# EPICS substitutions: iocs/example/labApp/Db/lab_expanded.substitutions
# This file was automatically generated on Fri 25 May 2018 08:06:14 BST from
# source: /home/hgv27681/R3.14.12.3/support/pmac/etc/makeIocs/lab.xml
#
# *** Please do not edit this file: edit the source file instead. ***
#

# Macros:
#  PORT      The asyn port for the pmac controller
#  P         PV Prefix
#  NAXES     Number of axes
#  TIMEOUT   Timeout for controller communication
#  FEEDRATE  feedrate below which we go into error
#  CSG0      Name for Coordinate System Group 0
#  CSG1      Name for Coordinate System Group 1
#  CSG2      Name for Coordinate System Group 2
#  CSG3      Name for Coordinate System Group 3
#  CSG4      Name for Coordinate System Group 4
#  CSG5      Name for Coordinate System Group 5
#  CSG6      Name for Coordinate System Group 6
#  CSG7      Name for Coordinate System Group 7
file $(PMAC)/db/pmacController.template
{
pattern { PORT, P, NAXES, TIMEOUT, FEEDRATE, CSG0, CSG1, CSG2, CSG3, CSG4, CSG5, CSG6, CSG7 }
    { "Brick", "BRICK1", "8", "4", "100", "1,2->A,B", "3,4->I", "MIXED CS3", "MIXED CS2", "", "", "", "" }
}

# Macros:
#  PORT  The asyn port for the pmac controller
#  P     PV Prefix
# For Non-Power PMAC, use pmacStatus.template instead
file $(PMAC)/db/powerPmacStatus.template
{
pattern { PORT, P }
    { "Brick", "BRICK1" }
}

# Macros:
#  PMAC  Pmac/Geobrick name
#  AXIS  Axis number
#  PORT  Asyn port
file $(PMAC)/db/pmacStatusAxis.template
{
pattern { PMAC, AXIS, PORT }
    { "BRICK1", "1", "Brick" }
    { "BRICK1", "2", "Brick" }
    { "BRICK1", "3", "Brick" }
    { "BRICK1", "4", "Brick" }
    { "BRICK1", "5", "Brick" }
    { "BRICK1", "6", "Brick" }
    { "BRICK1", "7", "Brick" }
    { "BRICK1", "8", "Brick" }
}

# Macros:
#  P                Device Prefix
#  M                Device Suffix
#  PORT             Delta tau motor controller
#  ADDR             Address on controller
#  DESC             Description, displayed on EDM screen
#  MRES             Motor Step Size (EGU)
#  VELO             Velocity (EGU/s)
#  PREC             Display Precision
#  EGU              Engineering Units
#  TWV              Tweak Step Size (EGU)
#  DTYP             DTYP of record
#  DIR              User Direction
#  VBAS             Base Velocity (EGU/s)
#  VMAX             Max Velocity (EGU/s), defaults to VELO
#  ACCL             Seconds to Velocity
#  BDST             BL Distance (EGU)
#  BVEL             BL Velocity (EGU/s)
#  BACC             BL Seconds to Veloc.
#  DHLM             Dial High Limit
#  DLLM             Dial Low Limit
#  HLM              User High Limit
#  LLM              User Low Limit
#  HLSV             HW Lim. Violation Svr
#  INIT             Startup commands
#  SREV             Steps per Revolution
#  RRES             Readback Step Size (EGU)
#  ERES             Encoder Step Size (EGU)
#  JAR              Jog Acceleration (EGU/s^2)
#  UEIP             Use Encoder If Present
#  URIP             Use RDBL If Present
#  RDBL             Readback Location, set URIP = 1 if you specify this
#  RLNK             Readback output link
#  RTRY             Max retry count
#  DLY              Readback settle time (s)
#  OFF              User Offset (EGU)
#  RDBD             Retry Deadband (EGU)
#  FOFF             Freeze Offset, 0=variable, 1=frozen
#  ADEL             Alarm monitor deadband (EGU)
#  NTM              New Target Monitor, only set to 0 for soft motors
#  FEHIGH           HIGH limit for following error
#  FEHIHI           HIHI limit for following error
#  FEHHSV           HIHI alarm severity for following error
#  FEHSV            HIGH alarm severity for following error
#  SCALE            Scale factor, if pmacSetAxisScale is used this should be set
#  HOMEVIS          If 1 then home is visible on the gui
#  HOMEVISSTR       If HOMEVIS=0, then display this text on the gui instead
#  name             Object name and gui association name
#  alh              Set this to alh to add the motor to the alarm handler and send emails,
#  gda_name         Name to export this as to GDA
#  gda_desc         Description to export this as to GDA
#  SPORT            Delta tau motor controller comms port
#  HOME             Prefix for autohome instance. Defaults to $(P). If unspecified,
#  ALLOW_HOMED_SET  Set to a blank to allow this axis to have its homed
file $(PMAC)/db/dls_pmac_asyn_motor.template
{
pattern { P, M, PORT, ADDR, DESC, MRES, VELO, PREC, EGU, TWV, DTYP, DIR, VBAS, VMAX, ACCL, BDST, BVEL, BACC, DHLM, DLLM, HLM, LLM, HLSV, INIT, SREV, RRES, ERES, JAR, UEIP, URIP, RDBL, RLNK, RTRY, DLY, OFF, RDBD, FOFF, ADEL, NTM, FEHIGH, FEHIHI, FEHHSV, FEHSV, SCALE, HOMEVIS, HOMEVISSTR, name, alh, gda_name, gda_desc, SPORT, HOME, PMAC, ALLOW_HOMED_SET }
    { "PMAC_BRICK_TEST", ":MOTOR1", "Brick", "1", "Motor 1->A", "1", "20", "3", "mm", "50", "asynMotor", "0", "0", "$(VELO)", "0.5", "0", "0", "", "10000", "-10000", "", "", "MAJOR", "", "1000", "", "", "", "0", "0", "", "", "0", "0", "0", "", "0", "0", "1", "0", "0", "NO_ALARM", "NO_ALARM", "1", "1", "Use motor summary screen", "M1", "None", "", "$(DESC)", "BRICK1port", "$(P)", "BRICK1", "#" }
    { "PMAC_BRICK_TEST", ":MOTOR2", "Brick", "2", "Motor 2->B", "1", "20", "3", "mm", "50", "asynMotor", "0", "0", "$(VELO)", "0.5", "0", "0", "", "10000", "-10000", "", "", "MAJOR", "", "1000", "", "", "", "0", "0", "", "", "0", "0", "0", "", "0", "0", "1", "0", "0", "NO_ALARM", "NO_ALARM", "1", "1", "Use motor summary screen", "M2", "None", "", "$(DESC)", "BRICK1port", "$(P)", "BRICK1", "#" }
    { "PMAC_BRICK_TEST", ":MOTOR3", "Brick", "3", "Motor 3->I JACK 1", "0.001", "20", "3", "mm", "50", "asynMotor", "0", "0", "$(VELO)", "0.5", "0", "0", "", "10000", "-10000", "", "", "MAJOR", "", "1000", "", "", "", "0", "0", "", "", "0", "0", "0", "", "0", "0", "1", "0", "0", "NO_ALARM", "NO_ALARM", "1", "1", "Use motor summary screen", "M3", "None", "", "$(DESC)", "BRICK1port", "$(P)", "BRICK1", "#" }
    { "PMAC_BRICK_TEST", ":MOTOR4", "Brick", "4", "Motor 4->I- JACK 2", "0.001", "20", "3", "mm", "50", "asynMotor", "0", "0", "$(VELO)", "0.5", "0", "0", "", "10000", "-10000", "", "", "MAJOR", "", "1000", "", "", "", "0", "0", "", "", "0", "0", "0", "", "0", "0", "1", "0", "0", "NO_ALARM", "NO_ALARM", "1", "1", "Use motor summary screen", "M4", "None", "", "$(DESC)", "BRICK1port", "$(P)", "BRICK1", "#" }
    { "PMAC_BRICK_TEST", ":MOTOR5", "Brick", "5", "Motor 5", "0.001", "20", "3", "mm", "10", "asynMotor", "0", "0", "$(VELO)", "0.5", "0", "0", "", "10000", "-10000", "", "", "MAJOR", "", "1000", "", "", "", "0", "0", "", "", "0", "0", "0", "", "0", "0", "1", "0", "0", "NO_ALARM", "NO_ALARM", "1", "1", "Use motor summary screen", "M5", "None", "", "$(DESC)", "BRICK1port", "$(P)", "BRICK1", "#" }
    { "PMAC_BRICK_TEST", ":MOTOR6", "Brick", "6", "Motor 6", "0.001", "20", "3", "mm", "10", "asynMotor", "0", "0", "$(VELO)", "0.5", "0", "0", "", "10000", "-10000", "", "", "MAJOR", "", "1000", "", "", "", "0", "0", "", "", "0", "0", "0", "", "0", "0", "1", "0", "0", "NO_ALARM", "NO_ALARM", "1", "1", "Use motor summary screen", "M6", "None", "", "$(DESC)", "BRICK1port", "$(P)", "BRICK1", "#" }
    { "PMAC_BRICK_TEST", ":MOTOR7", "Brick", "7", "Motor 7", "0.001", "20", "3", "mm", "10", "asynMotor", "0", "0", "$(VELO)", "0.5", "0", "0", "", "10000", "-10000", "", "", "MAJOR", "", "1000", "", "", "", "0", "0", "", "", "0", "0", "0", "", "0", "0", "1", "0", "0", "NO_ALARM", "NO_ALARM", "1", "1", "Use motor summary screen", "M7", "None", "", "$(DESC)", "BRICK1port", "$(P)", "BRICK1", "#" }
    { "PMAC_BRICK_TEST", ":MOTOR8", "Brick", "8", "Motor 8", "0.001", "20", "3", "mm", "10", "asynMotor", "0", "0", "$(VELO)", "0.5", "0", "0", "", "10000", "-10000", "", "", "MAJOR", "", "1000", "", "", "", "0", "0", "", "", "0", "0", "0", "", "0", "0", "1", "0", "0", "NO_ALARM", "NO_ALARM", "1", "1", "Use motor summary screen", "M8", "None", "", "$(DESC)", "BRICK1port", "$(P)", "BRICK1", "#" }
}

# Macros:
#  PORT     The asyn port for the pmac cs controller
#  PMAC     PV Prefix for the motor controller
#  CS       Coordinate System Number for the cs controller
#  TIMEOUT  Timeout for controller communication
file $(PMAC)/db/pmacCsController.template
{
pattern { PORT, PMAC, CS, TIMEOUT }
    { "CS1", "BRICK1", "1", "4" }
    { "CS2", "BRICK1", "2", "4" }
    { "CS3", "BRICK1", "3", "4" }
}

# Macros:
#  P           Device Prefix
#  M           Device Suffix
#  PORT        Delta tau motor controller
#  ADDR        Address on controller
#  DESC        Description, displayed on EDM screen
#  MRES        Motor Step Size (EGU)
#  VELO        Velocity (EGU/s)
#  PREC        Display Precision
#  EGU         Engineering Units
#  TWV         Tweak Step Size (EGU)
#  DTYP        DTYP of record
#  DIR         User Direction
#  VBAS        Base Velocity (EGU/s)
#  VMAX        Max Velocity (EGU/s), defaults to VELO
#  ACCL        Seconds to Velocity
#  BDST        BL Distance (EGU)
#  BVEL        BL Velocity (EGU/s)
#  BACC        BL Seconds to Veloc.
#  DHLM        Dial High Limit
#  DLLM        Dial Low Limit
#  HLM         User High Limit
#  LLM         User Low Limit
#  HLSV        HW Lim. Violation Svr
#  INIT        Startup commands
#  SREV        Steps per Revolution
#  RRES        Readback Step Size (EGU)
#  ERES        Encoder Step Size (EGU)
#  JAR         Jog Acceleration (EGU/s^2)
#  UEIP        Use Encoder If Present
#  URIP        Use RDBL If Present
#  RDBL        Readback Location, set URIP = 1 if you specify this
#  RLNK        Readback output link
#  RTRY        Max retry count
#  DLY         Readback settle time (s)
#  OFF         User Offset (EGU)
#  RDBD        Retry Deadband (EGU)
#  FOFF        Freeze Offset, 0=variable, 1=frozen
#  ADEL        Alarm monitor deadband (EGU)
#  NTM         New Target Monitor, only set to 0 for soft motors
#  FEHIGH      HIGH limit for following error
#  FEHIHI      HIHI limit for following error
#  FEHHSV      HIHI alarm severity for following error
#  FEHSV       HIGH alarm severity for following error
#  SCALE       Scale factor, if pmacSetAxisScale is used this should be set
#  HOMEVIS     If 1 then home is visible on the gui
#  HOMEVISSTR  If HOMEVIS=0, then display this text on the gui instead
#  name        Object name and gui association name
#  alh         Set this to alh to add the motor to the alarm handler and send emails,
#  gda_name    Name to export this as to GDA
#  gda_desc    Description to export this as to GDA
file $(PMAC)/db/dls_pmac_cs_asyn_motor.template
{
pattern { P, M, PORT, ADDR, DESC, MRES, VELO, PREC, EGU, TWV, DTYP, DIR, VBAS, VMAX, ACCL, BDST, BVEL, BACC, DHLM, DLLM, HLM, LLM, HLSV, INIT, SREV, RRES, ERES, JAR, UEIP, URIP, RDBL, RLNK, RTRY, DLY, OFF, RDBD, FOFF, ADEL, NTM, FEHIGH, FEHIHI, FEHHSV, FEHSV, SCALE, HOMEVIS, HOMEVISSTR, name, alh, gda_name, gda_desc, PMAC, CS }
    { "BRICK1CS2", ":A", "CS2", "1", "CS2 1->A", "0.0001", "20", "3", "mm", "1", "asynMotor", "0", "0", "$(VELO)", "0.5", "0", "0", "", "10000", "-10000", "", "", "MAJOR", "", "1000", "", "", "", "0", "0", "", "", "0", "0", "0", "", "0", "0", "1", "0", "0", "NO_ALARM", "NO_ALARM", "1", "1", "Use motor summary screen", "X2", "None", "", "$(DESC)", "BRICK1", "2" }
    { "BRICK1CS2", ":B", "CS2", "2", "CS2 2->B", "0.0001", "20", "3", "mm", "1", "asynMotor", "0", "0", "$(VELO)", "0.5", "0", "0", "", "10000", "-10000", "", "", "MAJOR", "", "1000", "", "", "", "0", "0", "", "", "0", "0", "0", "", "0", "0", "1", "0", "0", "NO_ALARM", "NO_ALARM", "1", "1", "Use motor summary screen", "Y2", "None", "", "$(DESC)", "BRICK1", "2" }
    { "BRICK1CS3", ":A", "CS3", "1", "CS3 1->A", "0.0001", "20", "3", "mm", "1", "asynMotor", "0", "0", "$(VELO)", "0.5", "0", "0", "", "10000", "-10000", "", "", "MAJOR", "", "1000", "", "", "", "0", "0", "", "", "0", "0", "0", "", "0", "0", "1", "0", "0", "NO_ALARM", "NO_ALARM", "1", "1", "Use motor summary screen", "A3", "None", "", "$(DESC)", "BRICK1", "3" }
    { "BRICK1CS3", ":B", "CS3", "2", "CS3 2->B", "0.0001", "20", "3", "mm", "1", "asynMotor", "0", "0", "$(VELO)", "0.5", "0", "0", "", "10000", "-10000", "", "", "MAJOR", "", "1000", "", "", "", "0", "0", "", "", "0", "0", "0", "", "0", "0", "1", "0", "0", "NO_ALARM", "NO_ALARM", "1", "1", "Use motor summary screen", "B3", "None", "", "$(DESC)", "BRICK1", "3" }
    { "BRICK1CS3", ":X", "CS3", "7", "CS3 HEIGHT", "0.0001", "20", "3", "mm", "1", "asynMotor", "0", "0", "$(VELO)", "0.5", "0", "0", "", "10000", "-10000", "", "", "MAJOR", "", "1000", "", "", "", "0", "0", "", "", "0", "0", "0", "", "0", "0", "1", "0", "0", "NO_ALARM", "NO_ALARM", "1", "1", "Use motor summary screen", "X3", "None", "", "$(DESC)", "BRICK1", "3" }
    { "BRICK1CS3", ":Y", "CS3", "8", "CS3 ANGLE", "0.0001", "20", "3", "deg", "1", "asynMotor", "0", "0", "$(VELO)", "0.5", "0", "0", "", "10000", "-10000", "", "", "MAJOR", "", "1000", "", "", "", "0", "0", "", "", "0", "0", "0", "", "0", "0", "1", "0", "0", "NO_ALARM", "NO_ALARM", "1", "1", "Use motor summary screen", "Y3", "None", "", "$(DESC)", "BRICK1", "3" }
}

# Macros:
#  PORT       Delta tau motor controller
#  NPOINTS    Number of points that can be built at any time
#  MAXPOINTS  Maximum number of points in a scan
#  PREC       precision of axis defnitions
file $(PMAC)/db/pmacControllerTrajectory.template
{
pattern { PORT, PMAC, NPOINTS, NAxes, MAXPOINTS, PREC }
    { "Brick", "BRICK1", "10000", "8", "4000000", "3" }
}

# Macros:
#  P           Pv Prefix
#  PLC         PLC number
#  PORT        Delta tau motor controller port
#  GRP1        Homing group 1 description
#  GRP2        Homing group 2 description
#  GRP3        Homing group 3 description
#  GRP4        Homing group 4 description
#  GRP5        Homing group 5 description
#  GRP6        Homing group 6 description
#  GRP7        Homing group 7 description
#  GRP8        Homing group 8 description
#  GRP9        Homing group 9 description
#  GRP10       Homing group 10 description
#  STATE11     Homing state 11 description
#  STATE12     Homing state 12 description
#  STATE13     Homing state 13 description
#  STATE14     Homing state 14 description
#  STATE15     Homing state 15 description
#  STATUS11    Homing status 11 description (e.g. for custom limit checks)
#  STATUS12    Homing status 12 description (e.g. for custom limit checks)
#  STATUS13    Homing status 13 description (e.g. for custom limit checks)
#  STATUS14    Homing status 14 description (e.g. for custom limit checks)
#  STATUS15    Homing status 15 description (e.g. for custom limit checks)
#  STATUSSV11  Homing status 11 severity
#  STATUSSV12  Homing status 12 severity
#  STATUSSV13  Homing status 13 severity
#  STATUSSV14  Homing status 14 severity
#  STATUSSV15  Homing status 15 severity
#  name        Object name and gui association name
#  DESC        Description
file $(PMAC)/db/autohome.template
{
pattern { P, PLC, PORT, CTRL, GRP1, GRP2, GRP3, GRP4, GRP5, GRP6, GRP7, GRP8, GRP9, GRP10, STATE11, STATE12, STATE13, STATE14, STATE15, STATUS11, STATUS12, STATUS13, STATUS14, STATUS15, STATUSSV11, STATUSSV12, STATUSSV13, STATUSSV14, STATUSSV15, name, DESC }
    { "PMAC_BRICK_TEST", "10", "Brick", "BRICK1", "All", "Axis1", "Axis2", "Axis3", "Axes4-8", "", "", "", "", "", "", "", "", "", "", "", "", "", "", "", "NO_ALARM", "NO_ALARM", "NO_ALARM", "NO_ALARM", "NO_ALARM", "HOME", "" }
}
